% RSLogix 500 project pH.RSS, saved by version 8.30.00.16 %
PROJECT "UNTITLED"    % processor: Bul.1763 MicroLogix 1100 Series B %

PROGRAM FILES
  LAD 2 "MAIN"  4 rungs
  LAD 3 "DIGITAL IO"  4 rungs
  LAD 4 "ANALOG IO"  4 rungs
  LAD 5 "CONTROLS"  4 rungs

DATA FILES
  O0 OUTPUT  7 elements
  I1 INPUT  13 elements
  S2 STATUS  66 elements
  B3 BINARY  1 elements
  T4 TIMER  2 elements
  C5 COUNTER  1 elements
  R6 CONTROL  1 elements
  N7 INTEGER  2 elements
  F8 FLOAT  1 elements
  PD9 PH  1 elements

LADDER 2 "MAIN"
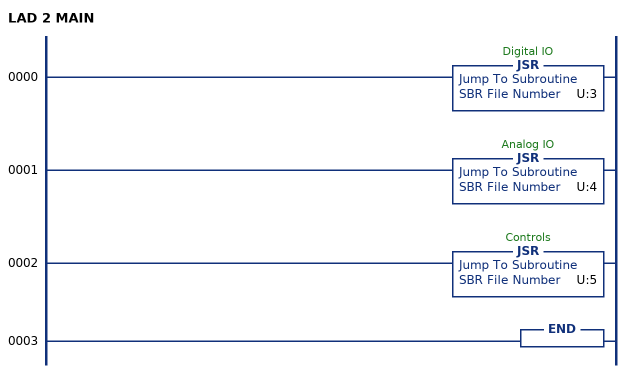
% Rung: 0 %
SOR JSR U:3 EOR
%   U:3  "Digital IO" %
% Rung: 1 %
SOR JSR U:4 EOR
%   U:4  "Analog IO" %
% Rung: 2 %
SOR JSR U:5 EOR
%   U:5  "Controls" %
% Rung: 3 %
SOR END EOR

LADDER 3 "DIGITAL IO"
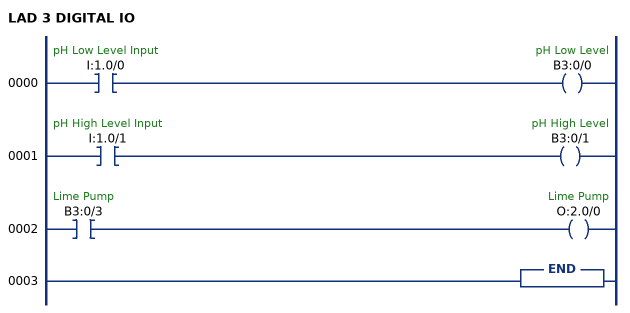
% Rung: 0 %
SOR XIC I:1.0/0 OTE B3:0/0 EOR
%   I:1.0/0  "pH Low Level Input" %
%   B3:0/0  "pH Low Level" %
% Rung: 1 %
SOR XIC I:1.0/1 OTE B3:0/1 EOR
%   I:1.0/1  "pH High Level Input" %
%   B3:0/1  "pH High Level" %
% Rung: 2 %
SOR XIC B3:0/3 OTE O:2.0/0 EOR
%   B3:0/3  "Lime Pump" %
%   O:2.0/0  "Lime Pump" %
% Rung: 3 %
SOR END EOR

LADDER 4 "ANALOG IO"
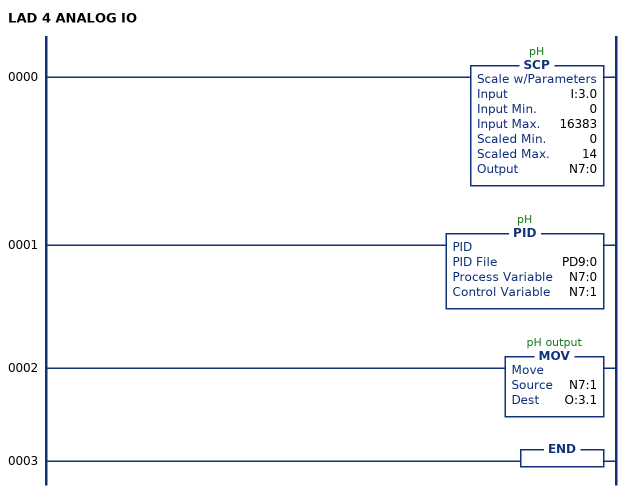
% Rung: 0 %
SOR SCP I:3.0 0 16383 0 14 N7:0 EOR
%   I:3.0  "pH Meter" %
%   N7:0  "pH" %
% Rung: 1 %
SOR PID PD9:0 N7:0 N7:1 EOR
%   PD9:0  "pH" %
%   N7:0  "pH" %
%   N7:1  "ph out" %
% Rung: 2 %
SOR MOV N7:1 O:3.1 EOR
%   N7:1  "ph out" %
%   O:3.1  "pH output" %
% Rung: 3 %
SOR END EOR

LADDER 5 "CONTROLS"
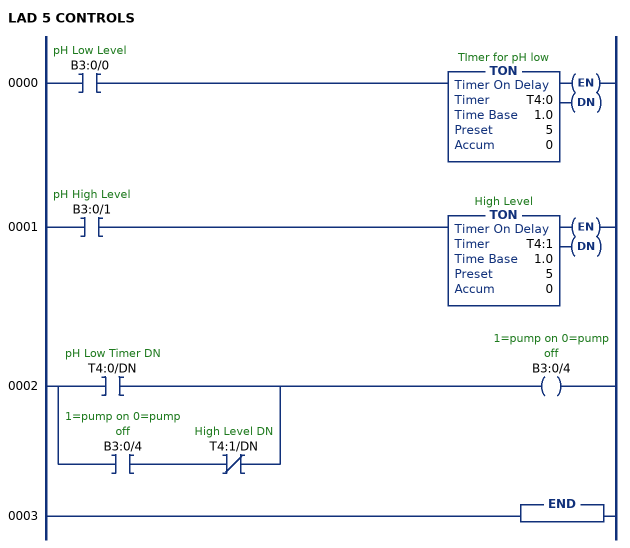
% Rung: 0 %
SOR XIC B3:0/0 TON T4:0 1.0 5 0 EOR
%   B3:0/0  "pH Low Level" %
%   T4:0  "TImer for pH low" %
% Rung: 1 %
SOR XIC B3:0/1 TON T4:1 1.0 5 0 EOR
%   B3:0/1  "pH High Level" %
%   T4:1  "High Level" %
% Rung: 2 %
SOR BST XIC T4:0/DN NXB XIC B3:0/4 XIO T4:1/DN BND OTE B3:0/4 EOR
%   T4:0/DN  "pH Low Timer DN" %
%   B3:0/4  "1=pump on 0=pump off" %
%   T4:1/DN  "High Level DN" %
% Rung: 3 %
SOR END EOR

OTHER DOCUMENTED ADDRESSES
  F8:0  "pH"
  F8:1  "pH PID Output"
  I:3.0/0  "pH Meter Reading"
  I:3.1  "pH Meter PID"
  O:2.0  LIME_PUMP  "Lime Pump"
  O:3.0/3  "out"
  O:3.3  "out"
  PD9  "pd9"

DATA TABLE (non-zero values as saved)
DATA T4
% .PRE .ACC %
% T4:0 % 5 0
% T4:1 % 5 0
